{attribute 'linkalways'} 
{attribute 'no_explicit_call' := 'This FB is a CLASS and must be accessed using methods or properties'}
{attribute 'enable_dynamic_creation'}
FUNCTION_BLOCK AlarmAddedEvent EXTENDS Disposable IMPLEMENTS I_AlarmAddedEvent
VAR
	_target : I_Alarm;
END_VAR

METHOD FB_init : BOOL
VAR_INPUT
	bInitRetains : BOOL; // if TRUE, the retain variables are initialized (warm start / cold start)
	bInCopyCode : BOOL;  // if TRUE, the instance afterwards gets moved into the copy code (online change)
	Target : I_Alarm;
END_VAR
This^._target := Target;
END_METHOD

PROPERTY PUBLIC Target : I_Alarm
GET
Target := _target;
END_GET
END_PROPERTY

END_FUNCTION_BLOCK

(* stored: Version 1.1.0.1, ProductVersion 3.1.4024.12
   POU AlarmAddedEvent: Id {6ded4ba6-036d-4378-bc08-3ce2b54f4581}, SpecialFunc None
   Folder Constructor: Id {b7f72a12-0b12-4dae-8d90-7bd07bd8c15d}
   Method FB_init: Id {7079e270-f3a7-418b-ac43-691c2a8748d5}
   Property Target: Id {3c0f6061-0116-4695-a000-e184031d4c6e}
   Get Get: Id {282e75d9-9697-4e0d-bdef-5453fa12cd09} *)
